FUNCTION_BLOCK EmergencyRecipeSequence (* Basic Function Block Type *)
  (* Standard: 61499-2 *)
  (* Version 0.0, 7/4/2026, Schneider Electric, Template *)
  PACKAGE SE.Nereda;
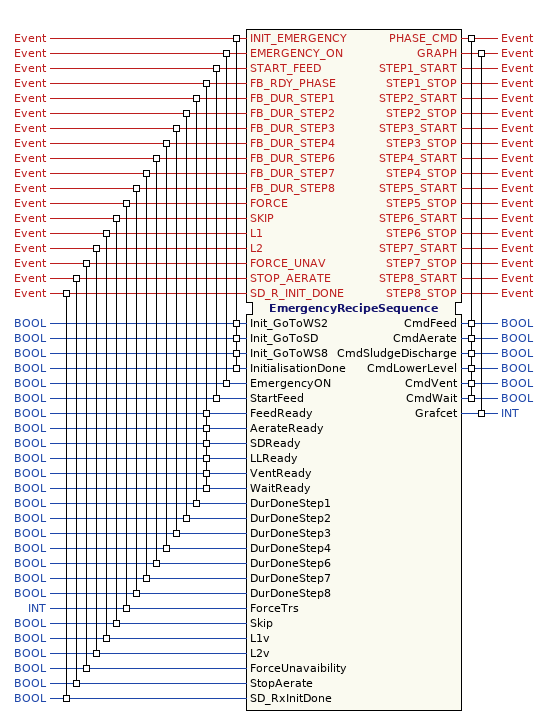
  EVENT_INPUT
    INIT_EMERGENCY WITH Init_GoToSD, Init_GoToWS8, InitialisationDone, Init_GoToWS2;
    EMERGENCY_ON WITH EmergencyON;
    START_FEED WITH StartFeed;
    FB_RDY_PHASE WITH FeedReady, AerateReady, SDReady, LLReady, VentReady, WaitReady;
    FB_DUR_STEP1 WITH DurDoneStep1;
    FB_DUR_STEP2 WITH DurDoneStep2;
    FB_DUR_STEP3 WITH DurDoneStep3;
    FB_DUR_STEP4 WITH DurDoneStep4;
    FB_DUR_STEP6 WITH DurDoneStep6;
    FB_DUR_STEP7 WITH DurDoneStep7;
    FB_DUR_STEP8 WITH DurDoneStep8;
    FORCE WITH ForceTrs;
    SKIP WITH Skip;
    L1 WITH L1v;
    L2 WITH L2v;
    FORCE_UNAV WITH ForceUnavaibility;
    STOP_AERATE WITH StopAerate;
    SD_R_INIT_DONE WITH SD_RxInitDone;
  END_EVENT
  EVENT_OUTPUT
    PHASE_CMD WITH CmdWait, CmdFeed, CmdAerate, CmdSludgeDischarge, CmdVent, CmdLowerLevel;
    GRAPH WITH Grafcet;
    STEP1_START;
    STEP1_STOP;
    STEP2_START;
    STEP2_STOP;
    STEP3_START;
    STEP3_STOP;
    STEP4_START;
    STEP4_STOP;
    STEP5_START;
    STEP5_STOP;
    STEP6_START;
    STEP6_STOP;
    STEP7_START;
    STEP7_STOP;
    STEP8_START;
    STEP8_STOP;
  END_EVENT
  VAR_INPUT
    Init_GoToWS2 : BOOL;
    Init_GoToSD : BOOL;
    Init_GoToWS8 : BOOL;
    InitialisationDone : BOOL;
    EmergencyON : BOOL;
    StartFeed : BOOL;
    FeedReady : BOOL;
    AerateReady : BOOL;
    SDReady : BOOL;
    LLReady : BOOL;
    VentReady : BOOL;
    WaitReady : BOOL;
    DurDoneStep1 : BOOL;
    DurDoneStep2 : BOOL;
    DurDoneStep3 : BOOL;
    DurDoneStep4 : BOOL;
    DurDoneStep6 : BOOL;
    DurDoneStep7 : BOOL;
    DurDoneStep8 : BOOL;
    ForceTrs : INT;
    Skip : BOOL;
    L1v : BOOL;
    L2v : BOOL;
    ForceUnavaibility : BOOL;
    StopAerate : BOOL;
    SD_RxInitDone : BOOL;
  END_VAR
  VAR_OUTPUT
    CmdFeed : BOOL;
    CmdAerate : BOOL;
    CmdSludgeDischarge : BOOL;
    CmdLowerLevel : BOOL;
    CmdVent : BOOL;
    CmdWait : BOOL;
    Grafcet : INT;
  END_VAR
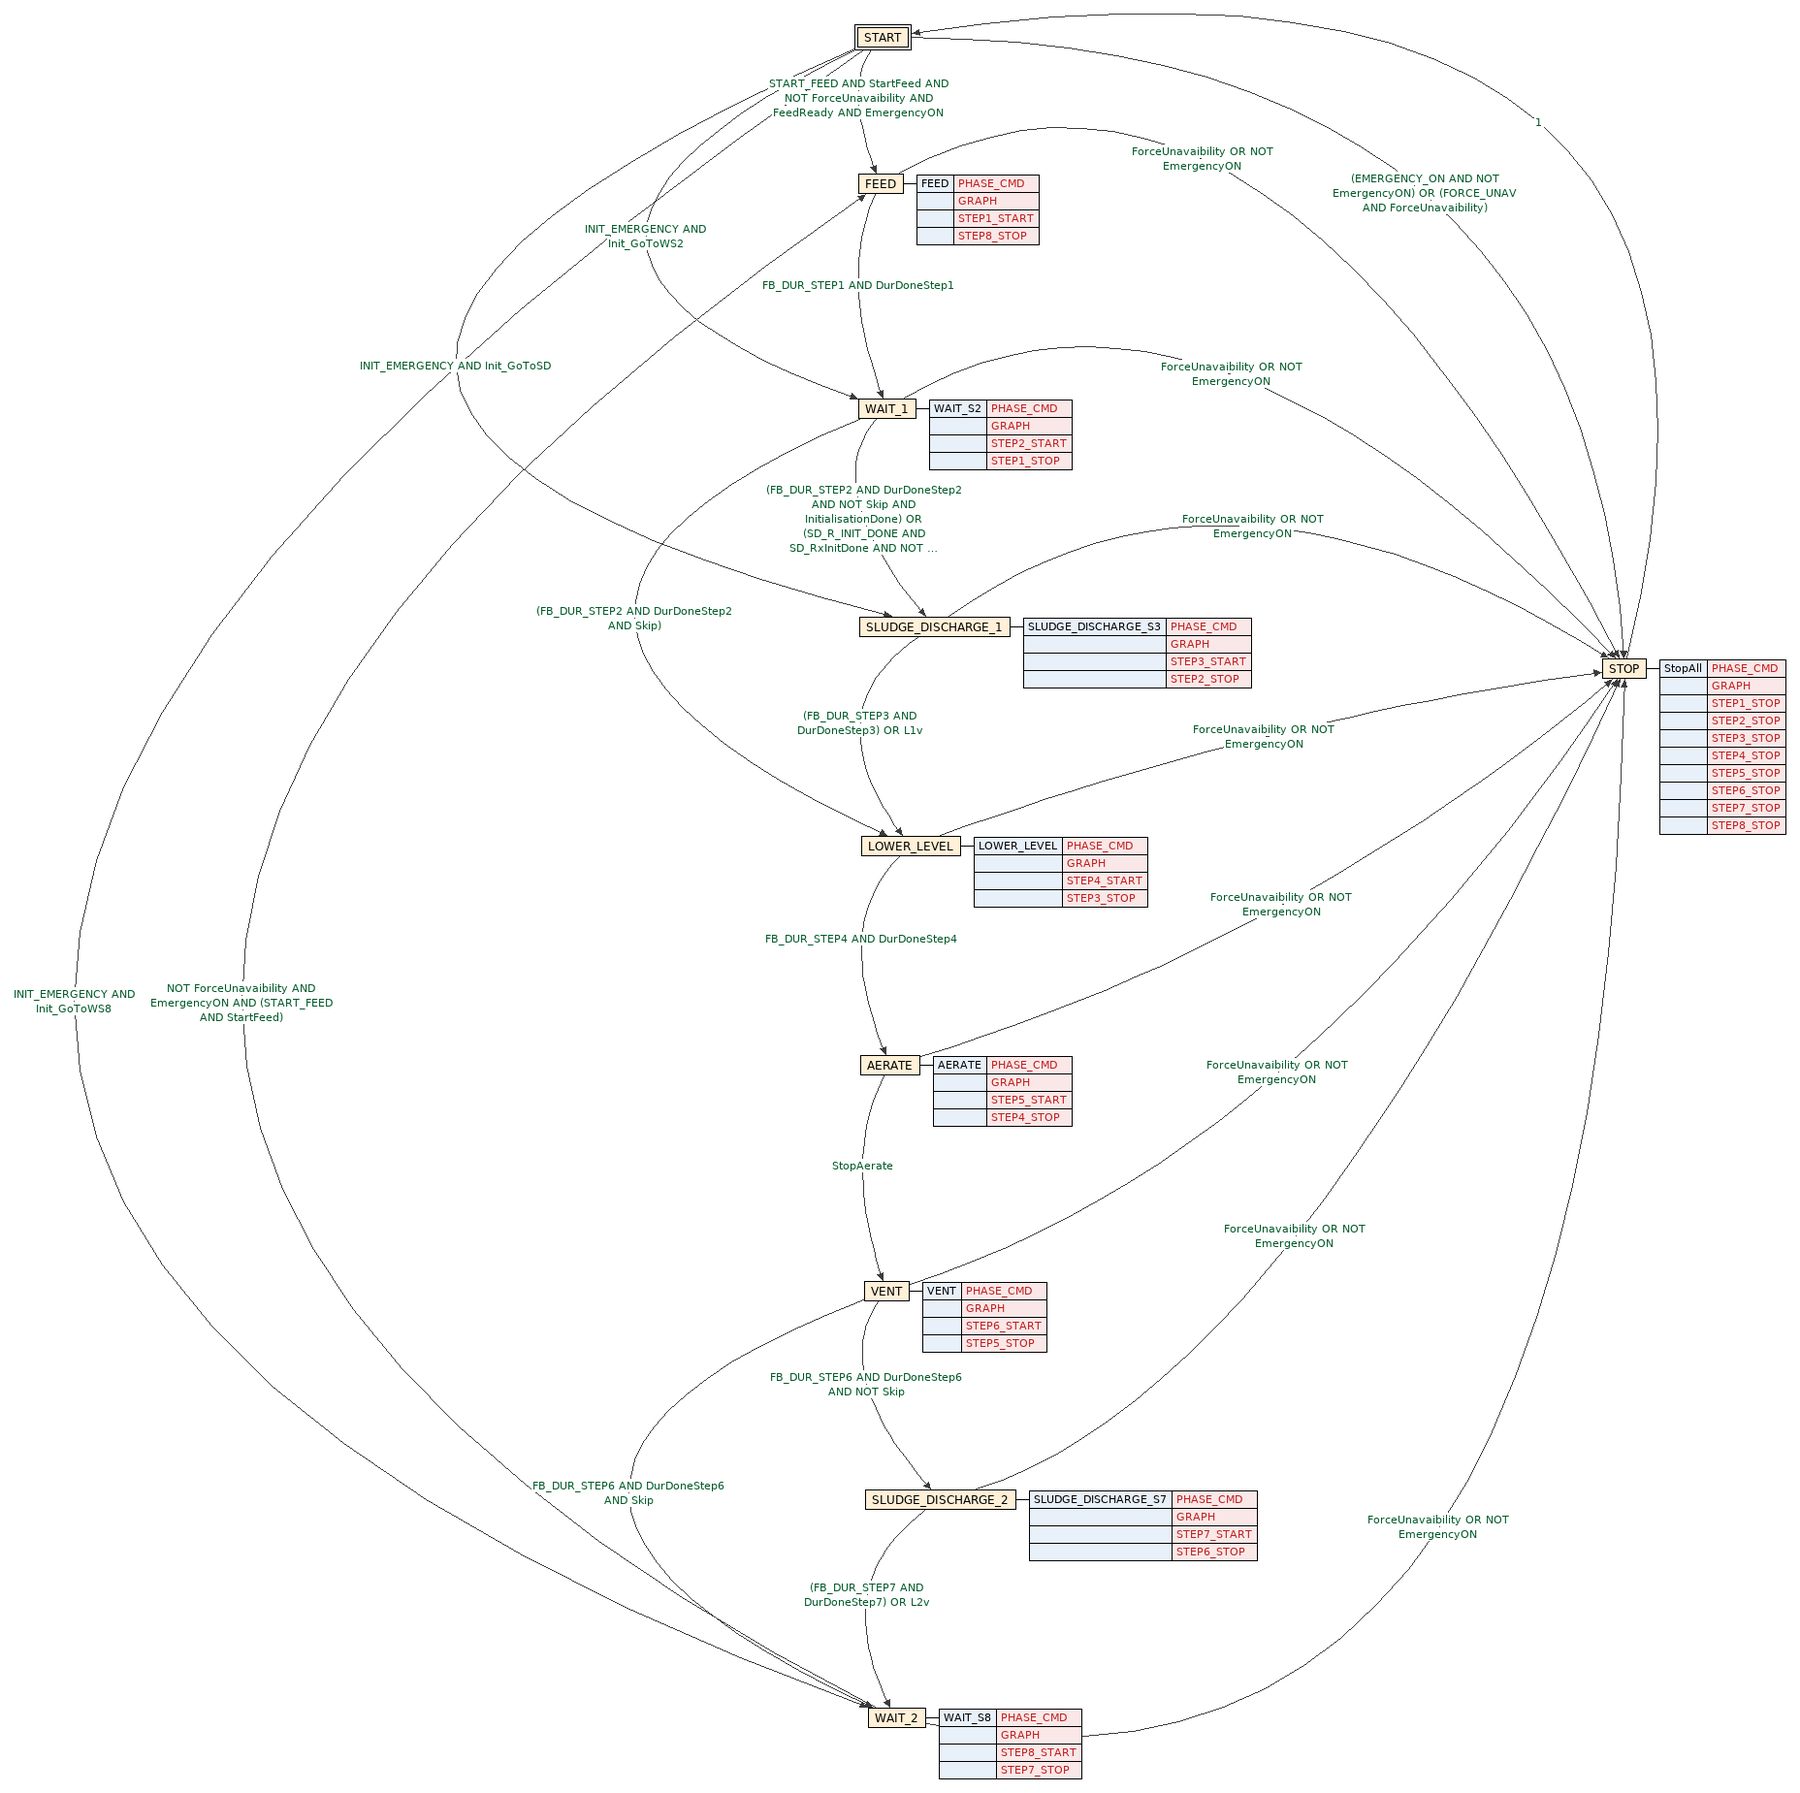
  EC_STATES
    START; (* Initial State *)
    FEED : FEED -> PHASE_CMD, -> GRAPH, -> STEP1_START, -> STEP8_STOP;
    WAIT_1 : WAIT_S2 -> PHASE_CMD, -> GRAPH, -> STEP2_START, -> STEP1_STOP;
    SLUDGE_DISCHARGE_1 : SLUDGE_DISCHARGE_S3 -> PHASE_CMD, -> GRAPH, -> STEP3_START, -> STEP2_STOP;
    LOWER_LEVEL : LOWER_LEVEL -> PHASE_CMD, -> GRAPH, -> STEP4_START, -> STEP3_STOP;
    AERATE : AERATE -> PHASE_CMD, -> GRAPH, -> STEP5_START, -> STEP4_STOP;
    VENT : VENT -> PHASE_CMD, -> GRAPH, -> STEP6_START, -> STEP5_STOP;
    SLUDGE_DISCHARGE_2 : SLUDGE_DISCHARGE_S7 -> PHASE_CMD, -> GRAPH, -> STEP7_START, -> STEP6_STOP;
    WAIT_2 : WAIT_S8 -> PHASE_CMD, -> GRAPH, -> STEP8_START, -> STEP7_STOP;
    STOP : StopAll -> PHASE_CMD, -> GRAPH, -> STEP1_STOP, -> STEP2_STOP, -> STEP3_STOP, -> STEP4_STOP, -> STEP5_STOP, -> STEP6_STOP, -> STEP7_STOP, -> STEP8_STOP;
  END_STATES
  EC_TRANSITIONS
    START TO FEED := START_FEED AND StartFeed AND NOT ForceUnavaibility AND FeedReady AND EmergencyON;
    FEED TO WAIT_1 := FB_DUR_STEP1 AND DurDoneStep1;
    WAIT_1 TO SLUDGE_DISCHARGE_1 := (FB_DUR_STEP2 AND DurDoneStep2 AND NOT Skip AND InitialisationDone) OR (SD_R_INIT_DONE AND SD_RxInitDone AND NOT InitialisationDone);
    SLUDGE_DISCHARGE_1 TO LOWER_LEVEL := (FB_DUR_STEP3 AND DurDoneStep3) OR L1v;
    LOWER_LEVEL TO AERATE := FB_DUR_STEP4 AND DurDoneStep4;
    AERATE TO VENT := StopAerate;
    VENT TO SLUDGE_DISCHARGE_2 := FB_DUR_STEP6 AND DurDoneStep6 AND NOT Skip;
    SLUDGE_DISCHARGE_2 TO WAIT_2 := (FB_DUR_STEP7 AND DurDoneStep7) OR L2v;
    START TO STOP := (EMERGENCY_ON AND NOT EmergencyON) OR (FORCE_UNAV AND ForceUnavaibility);
    STOP TO START := 1;
    FEED TO STOP := ForceUnavaibility OR NOT EmergencyON;
    WAIT_1 TO STOP := ForceUnavaibility OR NOT EmergencyON;
    SLUDGE_DISCHARGE_1 TO STOP := ForceUnavaibility OR NOT EmergencyON;
    LOWER_LEVEL TO STOP := ForceUnavaibility OR NOT EmergencyON;
    AERATE TO STOP := ForceUnavaibility OR NOT EmergencyON;
    VENT TO STOP := ForceUnavaibility OR NOT EmergencyON;
    SLUDGE_DISCHARGE_2 TO STOP := ForceUnavaibility OR NOT EmergencyON;
    WAIT_2 TO STOP := ForceUnavaibility OR NOT EmergencyON;
    WAIT_1 TO LOWER_LEVEL := (FB_DUR_STEP2 AND DurDoneStep2 AND Skip);
    VENT TO WAIT_2 := FB_DUR_STEP6 AND DurDoneStep6 AND Skip;
    START TO SLUDGE_DISCHARGE_1 := INIT_EMERGENCY AND Init_GoToSD;
    START TO WAIT_2 := INIT_EMERGENCY AND Init_GoToWS8;
    WAIT_2 TO FEED := NOT ForceUnavaibility AND EmergencyON AND (START_FEED AND StartFeed);
    START TO WAIT_1 := INIT_EMERGENCY AND Init_GoToWS2;
  END_TRANSITIONS
  ALGORITHM FEED IN ST:
;
CmdFeed := TRUE;
CmdAerate := FALSE;
CmdSludgeDischarge := FALSE;
CmdLowerLevel := FALSE;
CmdVent := FALSE;
CmdWait := FALSE;
Grafcet := 1;
  END_ALGORITHM
  ALGORITHM WAIT_S8 IN ST:
;
CmdFeed := FALSE;
CmdAerate := FALSE;
CmdSludgeDischarge := FALSE;
CmdLowerLevel := FALSE;
CmdVent := FALSE;
CmdWait := TRUE;

Grafcet := 8;
  END_ALGORITHM
  ALGORITHM SLUDGE_DISCHARGE_S7 IN ST:
;
CmdFeed := FALSE;
CmdAerate := FALSE;
CmdSludgeDischarge := TRUE;
CmdLowerLevel := FALSE;
CmdVent := FALSE;
CmdWait := FALSE;

Grafcet := 7;
  END_ALGORITHM
  ALGORITHM LOWER_LEVEL IN ST:
;
CmdFeed := FALSE;
CmdAerate := FALSE;
CmdSludgeDischarge := FALSE;
CmdLowerLevel := TRUE;
CmdVent := FALSE;
CmdWait := FALSE;
Grafcet := 4;
  END_ALGORITHM
  ALGORITHM AERATE IN ST:
;
CmdFeed := FALSE;
CmdAerate := TRUE;
CmdSludgeDischarge := FALSE;
CmdLowerLevel := FALSE;
CmdVent := FALSE;
CmdWait := FALSE;
Grafcet := 5;
  END_ALGORITHM
  ALGORITHM VENT IN ST:
;
CmdFeed := FALSE;
CmdAerate := FALSE;
CmdSludgeDischarge := FALSE;
CmdLowerLevel := FALSE;
CmdVent := TRUE;
CmdWait := FALSE;
Grafcet := 6;
  END_ALGORITHM
  ALGORITHM StopAll IN ST:
;
CmdFeed := FALSE;
CmdAerate := FALSE;
CmdSludgeDischarge := FALSE;
CmdLowerLevel := FALSE;
CmdVent := FALSE;
CmdWait := FALSE;
Grafcet := 10;
  END_ALGORITHM
  ALGORITHM Synchronize IN ST:
;
Grafcet := 9;
  END_ALGORITHM
  ALGORITHM WAIT_INIT IN ST:
;
CmdFeed := FALSE;
CmdAerate := FALSE;
CmdSludgeDischarge := FALSE;
CmdLowerLevel := FALSE;
CmdVent := FALSE;
CmdWait := TRUE;

Grafcet := 8;
  END_ALGORITHM
  ALGORITHM WAIT_S2 IN ST:
;
CmdFeed := FALSE;
CmdAerate := FALSE;
CmdSludgeDischarge := FALSE;
CmdLowerLevel := FALSE;
CmdVent := FALSE;
CmdWait := TRUE;

Grafcet := 2;
  END_ALGORITHM
  ALGORITHM SLUDGE_DISCHARGE_S3 IN ST:
;
CmdFeed := FALSE;
CmdAerate := FALSE;
CmdSludgeDischarge := TRUE;
CmdLowerLevel := FALSE;
CmdVent := FALSE;
CmdWait := FALSE;

Grafcet := 3;
  END_ALGORITHM
END_FUNCTION_BLOCK
